Staubli VAL3: oLid.pgx

public program oLid(num nChoice (dimensions=1))
// oLid
begin
  dioSet(oLid,nChoice)
end
